Fanuc KAREL source: kb00005.KL

-- PROVISIONAL review KL for V1013-1; original PC SHA256 d762813e8feafd52a0087bf9aa5cb422280bcb1ab75a01d8c19f5c40e27585a4
-- Incomplete behavior may be omitted. Consult companion uncertainty JSON. Do not deploy.
PROGRAM KB00005
%NOLOCKGROUP
BEGIN
  -- UNRESOLVED_PC offsets 5-14; opcodes 3F,75
  -- UNRESOLVED_PC offsets 19-28; opcodes 3F,75
  -- UNRESOLVED_PC offsets 33-42; opcodes 3F,75
  -- UNRESOLVED_PC offsets 47-54; opcodes 9D,23
  -- UNRESOLVED_PC offsets 59-66; opcodes 9D,23
  -- UNRESOLVED_PC offsets 71-111; opcodes 27,22,2A,22,2A,22,2A,22,22,31
  -- UNRESOLVED_PC offsets 116-120; opcodes 7F
END KB00005
